FUNCTION_BLOCK ADXL3x5Interface
VAR_INPUT
END_VAR
VAR_OUTPUT
END_VAR
VAR
END_VAR

END_FUNCTION_BLOCK

(* stored: Version 1.1.0.1, ProductVersion 3.1.4024.12
   POU ADXL3x5Interface: Id {c139e6f6-f214-44e8-9f0f-a559eda28c47}, SpecialFunc None *)
